// TIA Portal V17 export
// export: Created 2022-05-07T16:38:46.8875589Z, ExportSetting WithDefaults, DisplayName Totally Integrated Automation Portal, DisplayVersion V17 Update 3, DisplayName TIA Portal Openness, DisplayVersion V17 Update 3, DisplayName TIA Portal Version Control Interface, DisplayVersion V17, DisplayName TIA Portal Test Suite Advanced, DisplayVersion V17 Update 1, DisplayName SINAMICS Startdrive Advanced, DisplayVersion V17 Update2, DisplayName SINAMICS Startdrive G130, G150, S120, S150, SINAMICS MV, S210, DisplayVersion V17 Update2, DisplayName SINAMICS Startdrive G110M, G120, G120C, G120D, G120P, G115D, DisplayVersion V17 Update2, DisplayName STEP 7 Professional, DisplayVersion V17 Update 3, DisplayName STEP 7 Safety, DisplayVersion V17, DisplayName WinCC UA Professional, DisplayVersion V17 Update 3
DATA_BLOCK "FB_RIPRISTINO_MS_DB"   // DB16
VERSION : 0.1
// stored: AutoNumber true, DBAccessibleFromOPCUA true, InstanceOfName FB_RIPRISTINO_MS, InstanceOfType FB
"FB_RIPRISTINO_MS"
   // VAR_OUTPUT
   //    bDone : Bool;
   //    fase : Int;
   // END_VAR
   // VAR_IN_OUT
   //    bStart : Bool;
   // END_VAR
   // VAR
   //    T10 : TON_TIME;
   //    T35 : TON_TIME;
   // END_VAR
BEGIN
END_DATA_BLOCK
